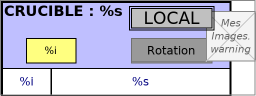
VISUALIZATION VISU_CREUSET  // 256x96
VAR_IN_OUT
	m_Input_CREUSET : BLOCK_IND_CR_396_TELEMARK;
END_VAR
VAR_INPUT
	m_Input_NUM_CRUCIBLE : SINT;
END_VAR
    Rectangle (1,1 230x95), "CRUCIBLE : %s", text variable: m_Input_NUM_CRUCIBLE
    RoundedRectangle (26,38 50x25), "%i", text variable: m_Input_CREUSET.PRM_NCR, invisible if: NOT Global_Variables.PRG_USER.ACTU_USER.MAINTENANCE OR NOT MACHINE.State_manu
        OnMouseDown: write the text variable via InputWithLimits, min 1, max 6
    Rectangle (51,68 179x27), "%s", text variable: m_Input_CREUSET.STATE_MAT
    Rectangle (2,68 49x27), "%i", text variable: m_Input_CREUSET.STATE_POS
    Button (131,38 81x25), "Rotation", colour toggle: m_Input_CREUSET.STATE_ROT, invisible if: NOT m_Input_CREUSET.AUTOR_Change_IHM OR NOT PRG_User.ACTU_USER.MAINTENANCE
        tap m_Input_CREUSET.M_Change
    Image (206,11 50x50), invisible if: NOT m_Input_CREUSET.State_nok, image: MesImages.warning
    RoundedRectangle (131,8 81x20), "REMOTE", invisible if: not m_Input_CREUSET.OUT_RMT
    RoundedRectangle (131,8 81x20), "LOCAL", invisible if: m_Input_CREUSET.OUT_RMT
    Rectangle (129,6 85x24), invisible if: Not m_Input_CREUSET.AUTOR_Remote_IHM, input disabled if: NOT PRG_User.ACTU_USER.MAINTENANCE
        tap m_Input_CREUSET.M_Remote
END_VISUALIZATION

(* stored: Version 1.1.0.1, ProductVersion 3.1.4026.18
   Visu VISU_CREUSET: Id {731f6e54-2ceb-4adc-af29-17e84b24dc19} *)
